(* PLC project SafeLOGIC-1, BrAutomation SafeDESIGNER  4.4.0.0 *)
(* stored: companyURL http://www.br-automation.com, creationDateTime Thu Jun 11 16:12:55 2020 *)

PROGRAM Main

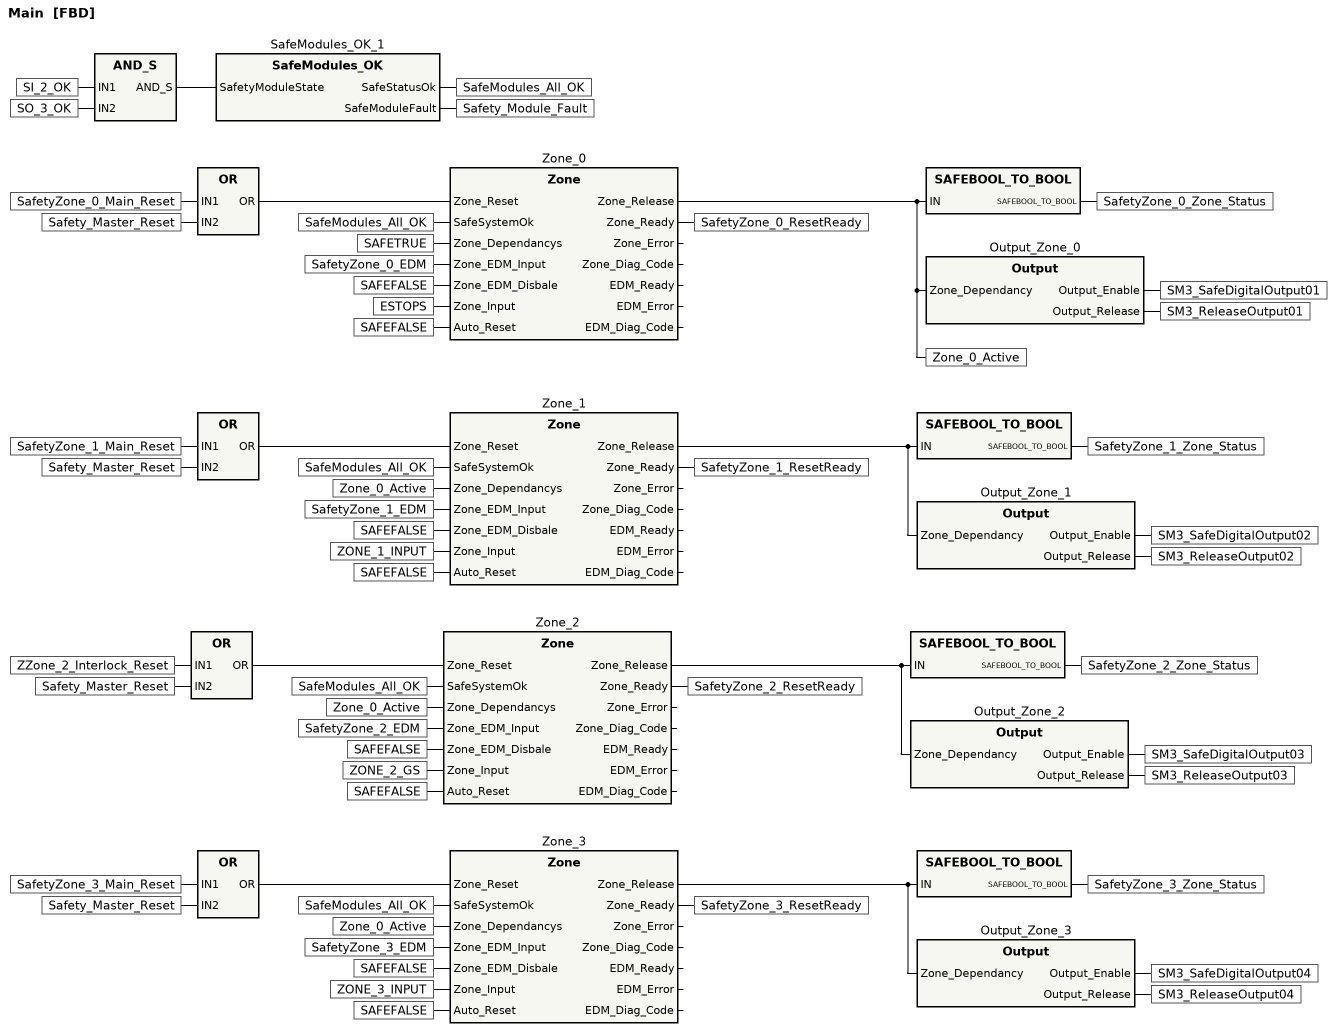
(* FBD diagram, written out as Structured Text *)
SafeModules_OK_1(SafetyModuleState := AND_S(SI_2_OK, SO_3_OK));
SafeModules_All_OK := SafeModules_OK_1.SafeStatusOk;
Safety_Module_Fault := SafeModules_OK_1.SafeModuleFault;
Zone_0(Zone_Reset := SafetyZone_0_Main_Reset OR Safety_Master_Reset, SafeSystemOk := SafeModules_All_OK, Zone_Dependancys := SAFETRUE, Zone_EDM_Input := SafetyZone_0_EDM, Zone_EDM_Disbale := SAFEFALSE, Zone_Input := ESTOPS, Auto_Reset := SAFEFALSE);
Zone_0_Active := Zone_0.Zone_Release;
SafetyZone_0_ResetReady := Zone_0.Zone_Ready;
SafetyZone_0_Zone_Status := SAFEBOOL_TO_BOOL(Zone_0.Zone_Release);
Output_Zone_0(Zone_Dependancy := Zone_0.Zone_Release);
SM3_SafeDigitalOutput01 := Output_Zone_0.Output_Enable;
SM3_ReleaseOutput01 := Output_Zone_0.Output_Release;
Zone_1(Zone_Reset := SafetyZone_1_Main_Reset OR Safety_Master_Reset, SafeSystemOk := SafeModules_All_OK, Zone_Dependancys := Zone_0_Active, Zone_EDM_Input := SafetyZone_1_EDM, Zone_EDM_Disbale := SAFEFALSE, Zone_Input := ZONE_1_INPUT, Auto_Reset := SAFEFALSE);
SafetyZone_1_ResetReady := Zone_1.Zone_Ready;
SafetyZone_1_Zone_Status := SAFEBOOL_TO_BOOL(Zone_1.Zone_Release);
Output_Zone_1(Zone_Dependancy := Zone_1.Zone_Release);
SM3_SafeDigitalOutput02 := Output_Zone_1.Output_Enable;
SM3_ReleaseOutput02 := Output_Zone_1.Output_Release;
Zone_2(Zone_Reset := ZZone_2_Interlock_Reset OR Safety_Master_Reset, SafeSystemOk := SafeModules_All_OK, Zone_Dependancys := Zone_0_Active, Zone_EDM_Input := SafetyZone_2_EDM, Zone_EDM_Disbale := SAFEFALSE, Zone_Input := ZONE_2_GS, Auto_Reset := SAFEFALSE);
SafetyZone_2_ResetReady := Zone_2.Zone_Ready;
SafetyZone_2_Zone_Status := SAFEBOOL_TO_BOOL(Zone_2.Zone_Release);
Output_Zone_2(Zone_Dependancy := Zone_2.Zone_Release);
SM3_SafeDigitalOutput03 := Output_Zone_2.Output_Enable;
SM3_ReleaseOutput03 := Output_Zone_2.Output_Release;
Zone_3(Zone_Reset := SafetyZone_3_Main_Reset OR Safety_Master_Reset, SafeSystemOk := SafeModules_All_OK, Zone_Dependancys := Zone_0_Active, Zone_EDM_Input := SafetyZone_3_EDM, Zone_EDM_Disbale := SAFEFALSE, Zone_Input := ZONE_3_INPUT, Auto_Reset := SAFEFALSE);
SafetyZone_3_ResetReady := Zone_3.Zone_Ready;
SafetyZone_3_Zone_Status := SAFEBOOL_TO_BOOL(Zone_3.Zone_Release);
Output_Zone_3(Zone_Dependancy := Zone_3.Zone_Release);
SM3_SafeDigitalOutput04 := Output_Zone_3.Output_Enable;
SM3_ReleaseOutput04 := Output_Zone_3.Output_Release;
END_PROGRAM
